Staubli VAL3: refreshStatic.pgx

program refreshStatic()
  local string l_sMenu
begin
  cls()
  //
  // set the view of the page..
  //
  // SET THE PAGE NUMBER
  use:nPage=0
  // USE <>PROFILE for <>PAGE
  use:nPage=use:nPage+abs(limit(global:mode,0,2)-2)
  // SET THE VIEW OF THE PAGE
  call language:page(l_sMenu,use:nPage)
  // define the menu
  call use:stringToArray(l_sMenu,sMenu)
  // set the menu
  call use:setMenu(sMenu,false,3)
  call use:getMenu(sMenu,bButton)
  //
  // CREATE THE LIST
  //
  // define your list size for default
  call use:setSizeList(17,0,21,10)
  call use:setView(bLarge)
  //
  call use:listcreate("")
  //
  call use:listadd(sList)
  //
  // refresh the cursor
  use:nView=nView
  // refresh the list
  call use:listupdate(nIndex-nView)
end
